FUNCTION_BLOCK FB_BumplessTransfer
VAR_INPUT
	u : ARRAY [0..5] OF LREAL;
	
	
	y_min : ARRAY [0..5] OF LREAL;
	y_max : ARRAY [0..5] OF LREAL;
	
END_VAR
VAR_OUTPUT
	y : ARRAY [0..5] OF LREAL;
END_VAR
VAR
	dof : UDINT;
END_VAR


// Saturate output
FOR dof := 0 TO 5 DO
	y[dof] := LIMIT(y_min[dof], u[dof], y_max[dof]);
END_FOR

METHOD FB_exit : BOOL
VAR_INPUT
	bInCopyCode : BOOL; // if TRUE, the exit method is called for exiting an instance that is copied afterwards (online change).
END_VAR
END_METHOD

METHOD FB_init : BOOL
VAR_INPUT
	bInitRetains : BOOL; // if TRUE, the retain variables are initialized (warm start / cold start)
	bInCopyCode : BOOL;  // if TRUE, the instance afterwards gets moved into the copy code (online change)
END_VAR
END_METHOD

METHOD FB_reinit : BOOL
VAR_INPUT
END_VAR
END_METHOD

END_FUNCTION_BLOCK

(* stored: Version 1.1.0.1, ProductVersion 3.1.4022.7
   POU FB_BumplessTransfer: Id {f7b493b0-16ad-411d-89d3-f35f18fc566a}, SpecialFunc None
   Method FB_exit: Id {035461f2-0c6f-44ac-9e70-63d3310ab04a}
   Method FB_init: Id {9dbfef8f-21b5-4deb-87c9-e30596487355}
   Method FB_reinit: Id {d26b8d75-f5b7-4d3d-a9e2-bb572116b2cd} *)
